{attribute 'qualified_only'}
VAR_GLOBAL
	iTest AT %I* : INT;
END_VAR

(* stored: Version 1.1.0.1, ProductVersion 3.1.4024.12
   GVL TEST: Id {65599d5c-dd91-47d2-a3a2-823ea159d2f5} *)
